FUNCTION_BLOCK FB_Convert_mA2Zisterne
VAR_INPUT
	iInput			:	INT;
	tRefresh		:	TIME;
END_VAR
VAR_OUTPUT
	wOutPerc		: WORD;
	wOutLiter		: WORD;
END_VAR
VAR
	iValueArith		: INT;
	iPercent		: REAL;
	iLiter			: REAL;
	tonBlock		: TON;
	fbArithMittel	: FB_ArithMittel10;
	i_finalValue	: INT;
	
	iMaxValofSensor : REAL := 20000;
	
	
END_VAR

tonBlock(IN := NOT tonBlock.Q, PT := tRefresh);

IF tonBlock.Q THEN
	
	fbArithMittel(iInputValue := iInput, iOut => iValueArith );
	
	//-------------------- Prozent ------------------------
	
	iPercent	:= (iValueArith / iMaxValofSensor) * 100;
	
	IF iPercent > 100 THEN
		iPercent := 100;
	END_IF
	
	//-----------------------------------------------------
	
	//-------------------- Liter --------------------------
	
	iLiter := (iPercent / 100) * 5000;
	
	//------------------------------------------------
	
	wOutPerc	:= REAL_TO_WORD(iPercent);
	wOutLiter	:= REAL_TO_WORD(iLiter);
	
END_IF

END_FUNCTION_BLOCK

(* stored: Version 1.1.0.1, ProductVersion 3.1.4024.4
   POU FB_Convert_mA2Zisterne: Id {8f17dd3d-7194-4910-a364-d341dc4d3a5b}, SpecialFunc None *)
